// TIA Portal V20 export
FUNCTION "01 T10 LANT Alarms" : Void   // FC1193, LAD
TITLE = ALARMS
{ S7_Optimized_Access := 'TRUE' }
// stored: AutoNumber false, IsIECCheckEnabled true, SetENOAutomatically false
   VAR_TEMP
      Trash : Bool;
   END_VAR
BEGIN

REGION Network 1: ============ ALARMS RESET ============
END_REGION

REGION Network 2: Alarms Reset
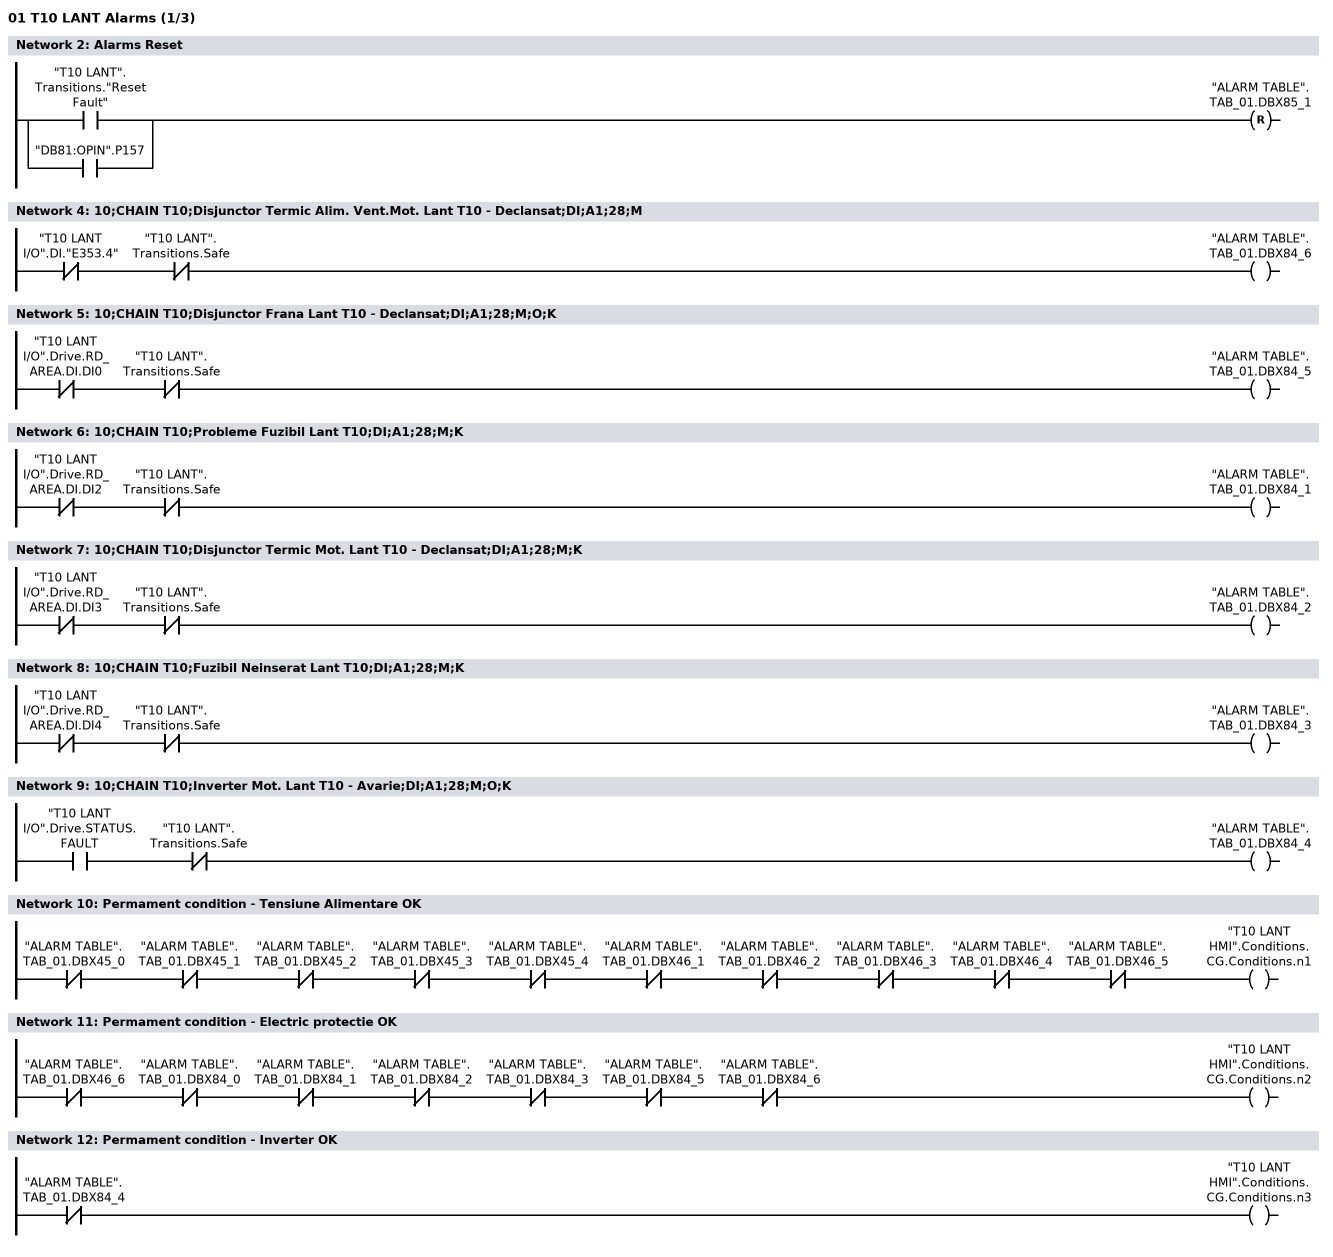
   RUNG wire#powerrail
      Contact( "T10 LANT".Transitions."Reset Fault" )
      wire#w1
      R_Coil( "ALARM TABLE".TAB_01.DBX85_1 )
   END_RUNG
   RUNG wire#powerrail
      Contact( "DB81:OPIN".P157 )
   END_RUNG wire#w1
   // the same network as SCL:
   IF "T10 LANT".Transitions."Reset Fault" OR "DB81:OPIN".P157 THEN
       "ALARM TABLE".TAB_01.DBX85_1 := FALSE;
   END_IF;
END_REGION

REGION Network 3: ============ PERMANENT CONDITIONS ============
END_REGION

REGION Network 4: 10;CHAIN T10;Disjunctor Termic Alim. Vent.Mot. Lant T10 - Declansat;DI;A1;28;M
   RUNG wire#powerrail
      I_Contact( "T10 LANT I/O".DI."E353.4" )
      I_Contact( "T10 LANT".Transitions.Safe )
      Coil( "ALARM TABLE".TAB_01.DBX84_6 )
   END_RUNG
   // the same network as SCL:
   "ALARM TABLE".TAB_01.DBX84_6 := NOT "T10 LANT I/O".DI."E353.4" AND NOT "T10 LANT".Transitions.Safe;
END_REGION

REGION Network 5: 10;CHAIN T10;Disjunctor Frana Lant T10 - Declansat;DI;A1;28;M;O;K
   RUNG wire#powerrail
      I_Contact( "T10 LANT I/O".Drive.RD_AREA.DI.DI0 )
      I_Contact( "T10 LANT".Transitions.Safe )
      Coil( "ALARM TABLE".TAB_01.DBX84_5 )
   END_RUNG
   // the same network as SCL:
   "ALARM TABLE".TAB_01.DBX84_5 := NOT "T10 LANT I/O".Drive.RD_AREA.DI.DI0 AND NOT "T10 LANT".Transitions.Safe;
END_REGION

REGION Network 6: 10;CHAIN T10;Probleme Fuzibil Lant T10;DI;A1;28;M;K
   RUNG wire#powerrail
      I_Contact( "T10 LANT I/O".Drive.RD_AREA.DI.DI2 )
      I_Contact( "T10 LANT".Transitions.Safe )
      Coil( "ALARM TABLE".TAB_01.DBX84_1 )
   END_RUNG
   // the same network as SCL:
   "ALARM TABLE".TAB_01.DBX84_1 := NOT "T10 LANT I/O".Drive.RD_AREA.DI.DI2 AND NOT "T10 LANT".Transitions.Safe;
END_REGION

REGION Network 7: 10;CHAIN T10;Disjunctor Termic Mot. Lant T10 - Declansat;DI;A1;28;M;K
   RUNG wire#powerrail
      I_Contact( "T10 LANT I/O".Drive.RD_AREA.DI.DI3 )
      I_Contact( "T10 LANT".Transitions.Safe )
      Coil( "ALARM TABLE".TAB_01.DBX84_2 )
   END_RUNG
   // the same network as SCL:
   "ALARM TABLE".TAB_01.DBX84_2 := NOT "T10 LANT I/O".Drive.RD_AREA.DI.DI3 AND NOT "T10 LANT".Transitions.Safe;
END_REGION

REGION Network 8: 10;CHAIN T10;Fuzibil Neinserat Lant T10;DI;A1;28;M;K
   RUNG wire#powerrail
      I_Contact( "T10 LANT I/O".Drive.RD_AREA.DI.DI4 )
      I_Contact( "T10 LANT".Transitions.Safe )
      Coil( "ALARM TABLE".TAB_01.DBX84_3 )
   END_RUNG
   // the same network as SCL:
   "ALARM TABLE".TAB_01.DBX84_3 := NOT "T10 LANT I/O".Drive.RD_AREA.DI.DI4 AND NOT "T10 LANT".Transitions.Safe;
END_REGION

REGION Network 9: 10;CHAIN T10;Inverter Mot. Lant T10 - Avarie;DI;A1;28;M;O;K
   RUNG wire#powerrail
      Contact( "T10 LANT I/O".Drive.STATUS.FAULT )
      I_Contact( "T10 LANT".Transitions.Safe )
      Coil( "ALARM TABLE".TAB_01.DBX84_4 )
   END_RUNG
   // the same network as SCL:
   "ALARM TABLE".TAB_01.DBX84_4 := "T10 LANT I/O".Drive.STATUS.FAULT AND NOT "T10 LANT".Transitions.Safe;
END_REGION

REGION Network 10: Permament condition - Tensiune Alimentare OK
   RUNG wire#powerrail
      I_Contact( "ALARM TABLE".TAB_01.DBX45_0 )
      I_Contact( "ALARM TABLE".TAB_01.DBX45_1 )
      I_Contact( "ALARM TABLE".TAB_01.DBX45_2 )
      I_Contact( "ALARM TABLE".TAB_01.DBX45_3 )
      I_Contact( "ALARM TABLE".TAB_01.DBX45_4 )
      I_Contact( "ALARM TABLE".TAB_01.DBX46_1 )
      I_Contact( "ALARM TABLE".TAB_01.DBX46_2 )
      I_Contact( "ALARM TABLE".TAB_01.DBX46_3 )
      I_Contact( "ALARM TABLE".TAB_01.DBX46_4 )
      I_Contact( "ALARM TABLE".TAB_01.DBX46_5 )
      Coil( "T10 LANT HMI".Conditions.CG.Conditions.n1 )
   END_RUNG
   // the same network as SCL:
   "T10 LANT HMI".Conditions.CG.Conditions.n1 := NOT "ALARM TABLE".TAB_01.DBX45_0 AND NOT "ALARM TABLE".TAB_01.DBX45_1 AND NOT "ALARM TABLE".TAB_01.DBX45_2 AND NOT "ALARM TABLE".TAB_01.DBX45_3 AND NOT "ALARM TABLE".TAB_01.DBX45_4 AND NOT "ALARM TABLE".TAB_01.DBX46_1 AND NOT "ALARM TABLE".TAB_01.DBX46_2 AND NOT "ALARM TABLE".TAB_01.DBX46_3 AND NOT "ALARM TABLE".TAB_01.DBX46_4 AND NOT "ALARM TABLE".TAB_01.DBX46_5;
END_REGION

REGION Network 11: Permament condition - Electric protectie OK
   RUNG wire#powerrail
      I_Contact( "ALARM TABLE".TAB_01.DBX46_6 )
      I_Contact( "ALARM TABLE".TAB_01.DBX84_0 )
      I_Contact( "ALARM TABLE".TAB_01.DBX84_1 )
      I_Contact( "ALARM TABLE".TAB_01.DBX84_2 )
      I_Contact( "ALARM TABLE".TAB_01.DBX84_3 )
      I_Contact( "ALARM TABLE".TAB_01.DBX84_5 )
      I_Contact( "ALARM TABLE".TAB_01.DBX84_6 )
      Coil( "T10 LANT HMI".Conditions.CG.Conditions.n2 )
   END_RUNG
   // the same network as SCL:
   "T10 LANT HMI".Conditions.CG.Conditions.n2 := NOT "ALARM TABLE".TAB_01.DBX46_6 AND NOT "ALARM TABLE".TAB_01.DBX84_0 AND NOT "ALARM TABLE".TAB_01.DBX84_1 AND NOT "ALARM TABLE".TAB_01.DBX84_2 AND NOT "ALARM TABLE".TAB_01.DBX84_3 AND NOT "ALARM TABLE".TAB_01.DBX84_5 AND NOT "ALARM TABLE".TAB_01.DBX84_6;
END_REGION

REGION Network 12: Permament condition - Inverter OK
   RUNG wire#powerrail
      I_Contact( "ALARM TABLE".TAB_01.DBX84_4 )
      Coil( "T10 LANT HMI".Conditions.CG.Conditions.n3 )
   END_RUNG
   // the same network as SCL:
   "T10 LANT HMI".Conditions.CG.Conditions.n3 := NOT "ALARM TABLE".TAB_01.DBX84_4;
END_REGION

REGION Network 13: Permanent condition
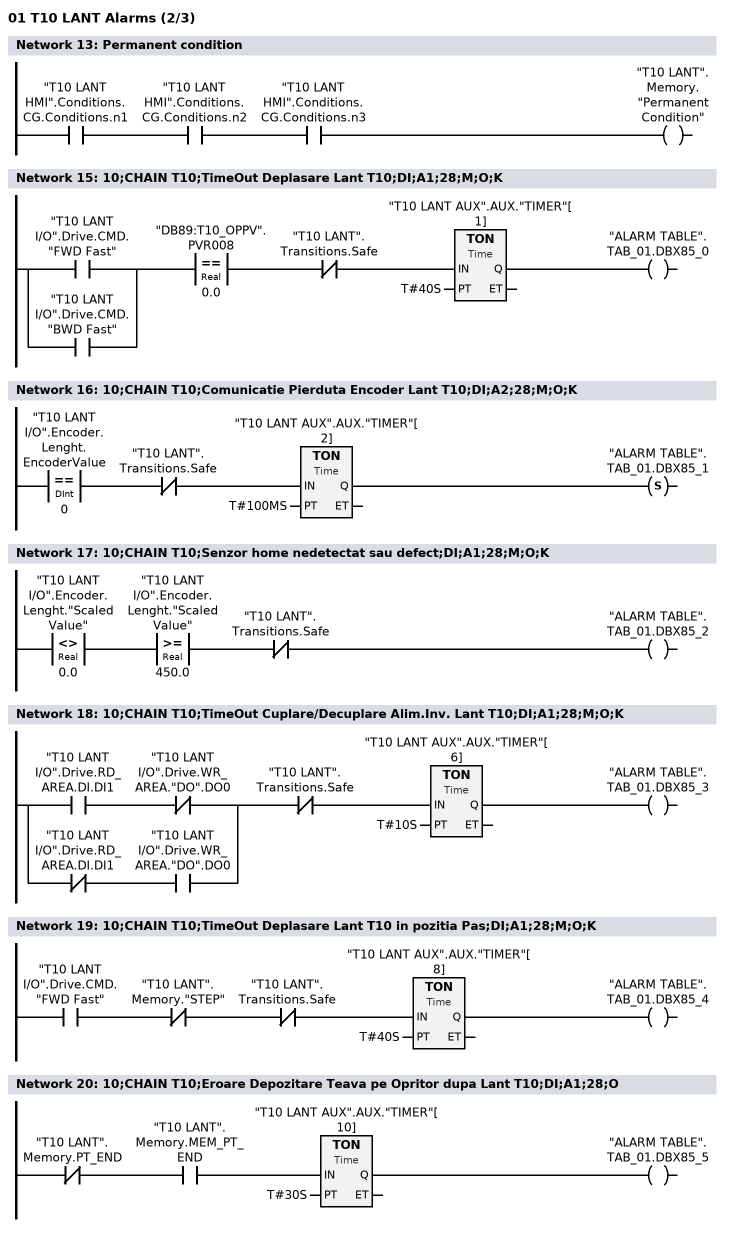
   RUNG wire#powerrail
      Contact( "T10 LANT HMI".Conditions.CG.Conditions.n1 )
      Contact( "T10 LANT HMI".Conditions.CG.Conditions.n2 )
      Contact( "T10 LANT HMI".Conditions.CG.Conditions.n3 )
      Coil( "T10 LANT".Memory."Permanent Condition" )
   END_RUNG
   // the same network as SCL:
   "T10 LANT".Memory."Permanent Condition" := "T10 LANT HMI".Conditions.CG.Conditions.n1 AND "T10 LANT HMI".Conditions.CG.Conditions.n2 AND "T10 LANT HMI".Conditions.CG.Conditions.n3;
END_REGION

REGION Network 14: ======= MACHINE MOVEMENT CONTROL (SENSORS / ENCODERS / INTERLOCKS) =======
END_REGION

REGION Network 15: 10;CHAIN T10;TimeOut Deplasare Lant T10;DI;A1;28;M;O;K
   RUNG wire#powerrail
      Contact( "T10 LANT I/O".Drive.CMD."FWD Fast" )
      wire#w1
      { S7_Templates := "SrcType := Real" } EQ_Contact(in1 := "DB89:T10_OPPV".PVR008, in2 := 0.0)
      I_Contact( "T10 LANT".Transitions.Safe )
      { S7_Templates := "time_type := Time" } "T10 LANT AUX".AUX."TIMER"[1].TON(pt := T#40S, et =>)
      Coil( "ALARM TABLE".TAB_01.DBX85_0 )
   END_RUNG
   RUNG wire#powerrail
      Contact( "T10 LANT I/O".Drive.CMD."BWD Fast" )
   END_RUNG wire#w1
   // the same network as SCL:
   "T10 LANT AUX".AUX."TIMER"[1].TON(IN := ("T10 LANT I/O".Drive.CMD."FWD Fast" OR "T10 LANT I/O".Drive.CMD."BWD Fast") AND ("DB89:T10_OPPV".PVR008 = 0.0) AND NOT "T10 LANT".Transitions.Safe,
                           PT := T#40S);
   "ALARM TABLE".TAB_01.DBX85_0 := "T10 LANT AUX".AUX."TIMER"[1].Q;
END_REGION

REGION Network 16: 10;CHAIN T10;Comunicatie Pierduta Encoder Lant T10;DI;A2;28;M;O;K
   RUNG wire#powerrail
      { S7_Templates := "SrcType := DInt" } EQ_Contact(in1 := "T10 LANT I/O".Encoder.Lenght.EncoderValue, in2 := 0)
      I_Contact( "T10 LANT".Transitions.Safe )
      { S7_Templates := "time_type := Time" } "T10 LANT AUX".AUX."TIMER"[2].TON(pt := T#100MS, et =>)
      S_Coil( "ALARM TABLE".TAB_01.DBX85_1 )
   END_RUNG
   // the same network as SCL:
   "T10 LANT AUX".AUX."TIMER"[2].TON(IN := ("T10 LANT I/O".Encoder.Lenght.EncoderValue = 0) AND NOT "T10 LANT".Transitions.Safe,
                           PT := T#100MS);
   IF "T10 LANT AUX".AUX."TIMER"[2].Q THEN "ALARM TABLE".TAB_01.DBX85_1 := TRUE; END_IF;
END_REGION

REGION Network 17: 10;CHAIN T10;Senzor home nedetectat sau defect;DI;A1;28;M;O;K
   RUNG wire#powerrail
      { S7_Templates := "SrcType := Real" } NE_Contact(in1 := "T10 LANT I/O".Encoder.Lenght."Scaled Value", in2 := 0.0)
      { S7_Templates := "SrcType := Real" } GE_Contact(in1 := "T10 LANT I/O".Encoder.Lenght."Scaled Value", in2 := 450.0)
      I_Contact( "T10 LANT".Transitions.Safe )
      Coil( "ALARM TABLE".TAB_01.DBX85_2 )
   END_RUNG
   // the same network as SCL:
   "ALARM TABLE".TAB_01.DBX85_2 := ("T10 LANT I/O".Encoder.Lenght."Scaled Value" <> 0.0) AND ("T10 LANT I/O".Encoder.Lenght."Scaled Value" >= 450.0) AND NOT "T10 LANT".Transitions.Safe;
END_REGION

REGION Network 18: 10;CHAIN T10;TimeOut Cuplare/Decuplare Alim.Inv. Lant T10;DI;A1;28;M;O;K
   RUNG wire#powerrail
      Contact( "T10 LANT I/O".Drive.RD_AREA.DI.DI1 )
      I_Contact( "T10 LANT I/O".Drive.WR_AREA."DO".DO0 )
      wire#w1
      I_Contact( "T10 LANT".Transitions.Safe )
      { S7_Templates := "time_type := Time" } "T10 LANT AUX".AUX."TIMER"[6].TON(pt := T#10S, et =>)
      Coil( "ALARM TABLE".TAB_01.DBX85_3 )
   END_RUNG
   RUNG wire#powerrail
      I_Contact( "T10 LANT I/O".Drive.RD_AREA.DI.DI1 )
      Contact( "T10 LANT I/O".Drive.WR_AREA."DO".DO0 )
   END_RUNG wire#w1
   // the same network as SCL:
   "T10 LANT AUX".AUX."TIMER"[6].TON(IN := (("T10 LANT I/O".Drive.RD_AREA.DI.DI1 AND NOT "T10 LANT I/O".Drive.WR_AREA."DO".DO0) OR (NOT "T10 LANT I/O".Drive.RD_AREA.DI.DI1 AND "T10 LANT I/O".Drive.WR_AREA."DO".DO0)) AND NOT "T10 LANT".Transitions.Safe,
                           PT := T#10S);
   "ALARM TABLE".TAB_01.DBX85_3 := "T10 LANT AUX".AUX."TIMER"[6].Q;
END_REGION

REGION Network 19: 10;CHAIN T10;TimeOut Deplasare Lant T10 in pozitia Pas;DI;A1;28;M;O;K
   RUNG wire#powerrail
      Contact( "T10 LANT I/O".Drive.CMD."FWD Fast" )
      I_Contact( "T10 LANT".Memory."STEP" )
      I_Contact( "T10 LANT".Transitions.Safe )
      { S7_Templates := "time_type := Time" } "T10 LANT AUX".AUX."TIMER"[8].TON(pt := T#40S, et =>)
      Coil( "ALARM TABLE".TAB_01.DBX85_4 )
   END_RUNG
   // the same network as SCL:
   "T10 LANT AUX".AUX."TIMER"[8].TON(IN := "T10 LANT I/O".Drive.CMD."FWD Fast" AND NOT "T10 LANT".Memory."STEP" AND NOT "T10 LANT".Transitions.Safe,
                           PT := T#40S);
   "ALARM TABLE".TAB_01.DBX85_4 := "T10 LANT AUX".AUX."TIMER"[8].Q;
END_REGION

REGION Network 20: 10;CHAIN T10;Eroare Depozitare Teava pe Opritor dupa Lant T10;DI;A1;28;O
   RUNG wire#powerrail
      I_Contact( "T10 LANT".Memory.PT_END )
      Contact( "T10 LANT".Memory.MEM_PT_END )
      { S7_Templates := "time_type := Time" } "T10 LANT AUX".AUX."TIMER"[10].TON(pt := T#30S, et =>)
      Coil( "ALARM TABLE".TAB_01.DBX85_5 )
   END_RUNG
   // the same network as SCL:
   "T10 LANT AUX".AUX."TIMER"[10].TON(IN := NOT "T10 LANT".Memory.PT_END AND "T10 LANT".Memory.MEM_PT_END,
                           PT := T#30S);
   "ALARM TABLE".TAB_01.DBX85_5 := "T10 LANT AUX".AUX."TIMER"[10].Q;
END_REGION

REGION Network 21: 10;CHAIN T10;TimeOut Cuplare/Decuplare Frana Lant T10;DI;A1;28;M;O;K
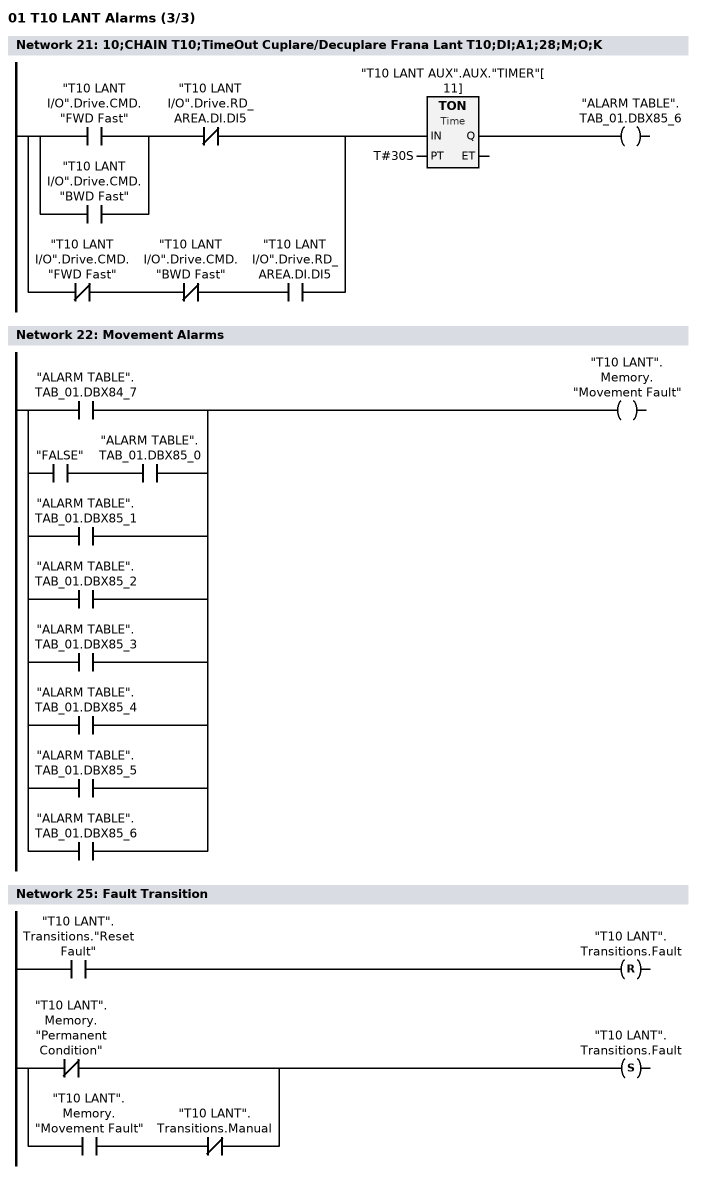
   RUNG wire#powerrail
      Contact( "T10 LANT I/O".Drive.CMD."FWD Fast" )
      wire#w1
      I_Contact( "T10 LANT I/O".Drive.RD_AREA.DI.DI5 )
      wire#w2
      { S7_Templates := "time_type := Time" } "T10 LANT AUX".AUX."TIMER"[11].TON(pt := T#30S, et =>)
      Coil( "ALARM TABLE".TAB_01.DBX85_6 )
   END_RUNG
   RUNG wire#powerrail
      Contact( "T10 LANT I/O".Drive.CMD."BWD Fast" )
   END_RUNG wire#w1
   RUNG wire#powerrail
      I_Contact( "T10 LANT I/O".Drive.CMD."FWD Fast" )
      I_Contact( "T10 LANT I/O".Drive.CMD."BWD Fast" )
      Contact( "T10 LANT I/O".Drive.RD_AREA.DI.DI5 )
   END_RUNG wire#w2
   // the same network as SCL:
   "T10 LANT AUX".AUX."TIMER"[11].TON(IN := (("T10 LANT I/O".Drive.CMD."FWD Fast" OR "T10 LANT I/O".Drive.CMD."BWD Fast") AND NOT "T10 LANT I/O".Drive.RD_AREA.DI.DI5) OR (NOT "T10 LANT I/O".Drive.CMD."FWD Fast" AND NOT "T10 LANT I/O".Drive.CMD."BWD Fast" AND "T10 LANT I/O".Drive.RD_AREA.DI.DI5),
                           PT := T#30S);
   "ALARM TABLE".TAB_01.DBX85_6 := "T10 LANT AUX".AUX."TIMER"[11].Q;
END_REGION

REGION Network 22: Movement Alarms
   RUNG wire#powerrail
      Contact( "ALARM TABLE".TAB_01.DBX84_7 )
      wire#w1
      Coil( "T10 LANT".Memory."Movement Fault" )
   END_RUNG
   RUNG wire#powerrail
      Contact( "FALSE" )
      Contact( "ALARM TABLE".TAB_01.DBX85_0 )
   END_RUNG wire#w1
   RUNG wire#powerrail
      Contact( "ALARM TABLE".TAB_01.DBX85_1 )
   END_RUNG wire#w1
   RUNG wire#powerrail
      Contact( "ALARM TABLE".TAB_01.DBX85_2 )
   END_RUNG wire#w1
   RUNG wire#powerrail
      Contact( "ALARM TABLE".TAB_01.DBX85_3 )
   END_RUNG wire#w1
   RUNG wire#powerrail
      Contact( "ALARM TABLE".TAB_01.DBX85_4 )
   END_RUNG wire#w1
   RUNG wire#powerrail
      Contact( "ALARM TABLE".TAB_01.DBX85_5 )
   END_RUNG wire#w1
   RUNG wire#powerrail
      Contact( "ALARM TABLE".TAB_01.DBX85_6 )
   END_RUNG wire#w1
   // the same network as SCL:
   "T10 LANT".Memory."Movement Fault" := "ALARM TABLE".TAB_01.DBX84_7 OR ("FALSE" AND "ALARM TABLE".TAB_01.DBX85_0) OR "ALARM TABLE".TAB_01.DBX85_1 OR "ALARM TABLE".TAB_01.DBX85_2 OR "ALARM TABLE".TAB_01.DBX85_3 OR "ALARM TABLE".TAB_01.DBX85_4 OR "ALARM TABLE".TAB_01.DBX85_5 OR "ALARM TABLE".TAB_01.DBX85_6;
END_REGION

REGION Network 23: ======= OTHER ALARMS =======
END_REGION

REGION Network 24: ======= FAULT =======
END_REGION

REGION Network 25: Fault Transition
   RUNG wire#powerrail
      Contact( "T10 LANT".Transitions."Reset Fault" )
      R_Coil( "T10 LANT".Transitions.Fault )
   END_RUNG
   RUNG wire#powerrail
      I_Contact( "T10 LANT".Memory."Permanent Condition" )
      wire#w1
      S_Coil( "T10 LANT".Transitions.Fault )
   END_RUNG
   RUNG wire#powerrail
      Contact( "T10 LANT".Memory."Movement Fault" )
      I_Contact( "T10 LANT".Transitions.Manual )
   END_RUNG wire#w1
   // the same network as SCL:
   IF "T10 LANT".Transitions."Reset Fault" THEN "T10 LANT".Transitions.Fault := FALSE; END_IF;
   IF NOT "T10 LANT".Memory."Permanent Condition" OR ("T10 LANT".Memory."Movement Fault" AND NOT "T10 LANT".Transitions.Manual) THEN
       "T10 LANT".Transitions.Fault := TRUE;
   END_IF;
END_REGION
END_FUNCTION
